FUNCTION_BLOCK cfbTest (* Composite Function Block Type *)
  (* Standard: 61499-2 *)
  (* Version 0.0, 10/2/2026, Schneider Electric, template *)
  PACKAGE Main;
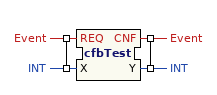
  EVENT_INPUT
    REQ WITH X; (* Normal Execution Request *)
  END_EVENT
  EVENT_OUTPUT
    CNF WITH Y; (* Execution Confirmation *)
  END_EVENT
  VAR_INPUT
    X : INT;
  END_VAR
  VAR_OUTPUT
    Y : INT;
  END_VAR
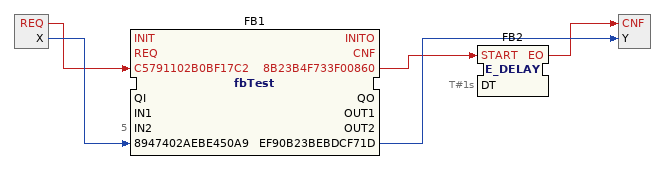
  FBS
    FB1 : fbTest(IN2 := 5);
    FB2 : E_DELAY(DT := T#1s);
  END_FBS
  EVENT_CONNECTIONS
    REQ TO FB1.C5791102B0BF17C2;
    FB2.EO TO CNF;
    FB1.8B23B4F733F00860 TO FB2.START;
  END_CONNECTIONS
  DATA_CONNECTIONS
    X TO FB1.8947402AEBE450A9;
    FB1.EF90B23BEBDCF71D TO Y;
  END_CONNECTIONS
END_FUNCTION_BLOCK
